FUNCTION_BLOCK StrapMachine
VAR_OUTPUT
	error AT %I* : BOOL;
	ready AT %I* : BOOL;
	busy AT %I* : BOOL;
	done (*AT %I**) : BOOL;
	home AT %I* : BOOL;
	
	execute AT %Q* : BOOL;
	enable AT %Q* : BOOL;
	reset AT %Q* : BOOL;
	
	timeout : BOOL;
END_VAR
VAR
	topSuction AT %Q* : BOOL;
	bottomSuction AT %Q* : BOOL;
	
	holdPost : TON;
	delay : TON;
	
	step : (SETUP, RUN, WAIT);
END_VAR
VAR_STAT CONSTANT
	pulseTime : TIME := T#100MS;
	holdTime : TIME := T#500MS;
	maxDelay : TIME := T#30S;
END_VAR

holdPost(IN:= , PT:= holdTime, Q=> , ET=> );
delay(IN:= step > 0, PT:= maxDelay, Q=> , ET=> );

IF delay.Q THEN
	delay.IN := FALSE;
	timeout := TRUE;
	
	step := SETUP;
END_IF

CASE step OF
	SETUP:
		busy := FALSE;
		IF error THEN
			reset := NOT reset;
			enable := FALSE;//NOT enable;
			
		ELSE
			reset := FALSE;
			enable := TRUE;
			
		END_IF
	
	RUN:
		IF NOT execute THEN
			execute := TRUE;
			RETURN;
		END_IF
		
		IF execute AND NOT home AND busy THEN
			execute := FALSE;
			step := WAIT;
		END_IF
		
	WAIT:
		IF home THEN
			holdPost.IN := TRUE;
			enable := FALSE;
			execute := FALSE;
		END_IF
		
		IF holdPost.Q THEN
			holdPost.IN := FALSE;
			done := TRUE;
			step := 0;
		END_IF
		
END_CASE

(*
executePulse(IN:= , PT:= pulseTime, Q=> , ET=> );
execute := executePulse.IN AND NOT executePulse.Q;

IF executePulse.Q THEN
	executePulse.IN := FALSE;
END_IF


resetPulse(IN:= , PT:= pulseTime, Q=> , ET=> );
StrapMachineST.reset := resetPulse.IN AND NOT resetPulse.Q;

IF resetPulse.Q THEN
	executePulse.IN := FALSE;
END_IF

ready := enable AND NOT execute AND NOT StrapMachineST.reset AND NOT error AND home;
*)

METHOD clear : BOOL
VAR_INPUT
END_VAR
(*
reset should be continuously called until machine returns evidence that it is ready again
machine is expected to not respond to reset signals if it is already in an idle state
*)
enable := FALSE;
execute := FALSE;

IF error THEN
	reset := NOT reset;
	clear := NOT error;

ELSE
	reset := FALSE;
	clear := TRUE;
	
END_IF
END_METHOD

METHOD strap : BOOL
VAR_INPUT
END_VAR
step := RUN;
END_METHOD

END_FUNCTION_BLOCK

(* stored: Version 1.1.0.1, ProductVersion 3.1.4024.11
   POU StrapMachine: Id {77eca895-fb38-4b31-8c37-4dfd9530abc9}, SpecialFunc None
   Method clear: Id {546729f9-8aa6-4691-b629-8aaf28ac27b0}
   Method strap: Id {bbf50787-b85f-4218-b3ad-09732c40ad08} *)
